PROGRAM P_SerialCom
VAR
	(*テストではパソコンにシリアルポートが無いので未使用
	fbModbusRtuSlave_PcCOM			:ModbusRtuSlave_PcCOM;
	*)
	
	//テスト用のファンクションブロック
	fbSerialLineControlADS				:SerialLineControlADS;
	fbModbusRtuSlave_Generic			:ModbusRtuSlave_Generic;
	
	//テスト用の変数
	bConnect							:BOOL:=TRUE;
	stSerialCfg							:ComSerialConfig;
	RxBuffer							:ComBuffer;
	TxBuffer							:ComBuffer;
	bAdsError							:BOOL;
	nAdsErrorID							:UDINT;	

END_VAR

//----テスト用のModbus通信---
	//シリアル接続を設定
	stSerialCfg.ComPort			:=3;
	stSerialCfg.Baudrate		:=9600;
	stSerialCfg.Parity			:=PARITY_NONE;
	stSerialCfg.DataBits		:=8;
	stSerialCfg.StopBits		:=STOPBITS_ONE;
	stSerialCfg.DTR				:=DTR_CTRL_DISABLE;
	stSerialCfg.RTS				:=RTS_CTRL_DISABLE;
	stSerialCfg.CTS				:=FALSE;
	stSerialCfg.DSR				:=FALSE;
	
	//USB接続のシリアルポートで通信
	fbSerialLineControlADS(	Connect		:=bConnect,
							SerialCfg	:=stSerialCfg,
							NetId		:='192.168.15.15.1.1',
							Timeout		:=DEFAULT_ADS_TIMEOUT,
							TxBuffer	:=TxBuffer,
							RxBuffer	:=RxBuffer,
							PortOpened	=>,
							Error		=>bAdsError,
							ErrorID		=>nAdsErrorID,
							Busy		=>,
							TxBufCount	=>,
							RxBufCount	=>
							);
	
	//Modbus通信
	fbModbusRtuSlave_Generic(	UnitID				:=1,
								AdrInputs			:=ADR(GVL_SerialCom.Inputs),
								SizeInputBytes		:=SIZEOF(GVL_SerialCom.Inputs),
								AdrOutputs			:=ADR(GVL_SerialCom.Outputs),
								SizeOutputBytes		:=SIZEOF(GVL_SerialCom.Outputs),
								AdrMemory			:=ADR(GVL_SerialCom.Memory),
								SizeMemoryBytes		:=SIZEOF(GVL_SerialCom.Memory),
								RxBuffer			:=RxBuffer,
								TxBuffer			:=TxBuffer,
								ErrorId				=>
								);

END_PROGRAM

(* stored: Version 1.1.0.1
   POU P_SerialCom: Id {b19f171e-24a4-40f9-86b0-32983ede39fc}, SpecialFunc None *)
